// TIA Portal project "fill_level_inspector_1st_stage" (V17)

(* hardware
DEVICE "S7-1200 station_1"  S7-1200 Station
   slot 0: "Rack_0"  S7-1200 Rack  Rack  V1.0
   slot 1: "PLC_1"  CPU 1212C AC/DC/Rly  6ES7 212-1BE31-0XB0  V3.0
   slot 2: "DI 16x24VDC/DQ 16xRelay_1"  SM 1223 DI16/DQ16 x relay  6ES7 223-1PL32-0XB0  V2.0
DEVICE "HMI_1"  KTP600 Basic color PN
   slot 0: "HMI_1"  KTP600 Basic color PN  6AV6 647-0AD11-3AX0  12.0.0.0
   slot 1: "HMI_RT_1"  KTP600 Basic color PN  6AV6 647-0AD11-3AX0  12.0.0.0
   slot 5: "HMI_1.IE_CP_1"  PROFINET Interface  12.0.0.0
      slot 1: "PROFINET Interface_1"  PROFINET Interface
         slot 1: "Port_1"  Port
*)

// ===== PLC "PLC_1"  CPU 1212C AC/DC/Rly =====

VAR_GLOBAL   // PLC tag table "Default tag table"
   "START" AT %M0.0 : Bool;
   "STOP" AT %M0.1 : Bool;
   "SYSTEM_RUN" AT %M0.2 : Bool;
   "Bottle_Animation" AT %MW20 : Int;
   "Bottle_Output" AT %M50.0 : Bool;
   "Filling_Animation" AT %MW22 : Int;
   "Filling_Output" AT %M50.1 : Bool;
   "BottleFull_Animation" AT %MW24 : Int;
   "BottleFull_Output" AT %M50.2 : Bool;
   "Clock_Byte" AT %MB100 : Byte;
   "Clock_10Hz" AT %M100.0 : Bool;
   "Clock_5Hz" AT %M100.1 : Bool;
   "Clock_2.5Hz" AT %M100.2 : Bool;
   "Clock_2Hz" AT %M100.3 : Bool;
   "Clock_1.25Hz" AT %M100.4 : Bool;
   "Clock_1Hz" AT %M100.5 : Bool;
   "Clock_0.625Hz" AT %M100.6 : Bool;
   "Clock_0.5Hz" AT %M100.7 : Bool;
END_VAR

// folder: System blocks/Program resources

DATA_BLOCK "Counter_Bottle_Animation"   // DB1
{ S7_Optimized_Access := 'TRUE' }
AUTHOR : Simatic
FAMILY : IEC
NAME : CNTR
VERSION : 1.0
// stored: InstanceOfName IEC_COUNTER
"IEC_COUNTER"
BEGIN
END_DATA_BLOCK

DATA_BLOCK "Counter_Filling_Animation"   // DB4
{ S7_Optimized_Access := 'TRUE' }
AUTHOR : Simatic
FAMILY : IEC
NAME : CNTR
VERSION : 1.0
// stored: InstanceOfName IEC_COUNTER
"IEC_COUNTER"
BEGIN
END_DATA_BLOCK

DATA_BLOCK "Counter_BottleFull_Animation"   // DB5
{ S7_Optimized_Access := 'TRUE' }
AUTHOR : Simatic
FAMILY : IEC
NAME : CNTR
VERSION : 1.0
// stored: InstanceOfName IEC_COUNTER
"IEC_COUNTER"
BEGIN
END_DATA_BLOCK

// folder: (top level)

ORGANIZATION_BLOCK "Main"   // OB1, LAD, ProgramCycle
TITLE = "Main Program Sweep (Cycle)"
{ S7_Optimized_Access := 'TRUE' }
VERSION : 0.1
BEGIN

REGION Network 1: OPEN/CLOSE VALVE
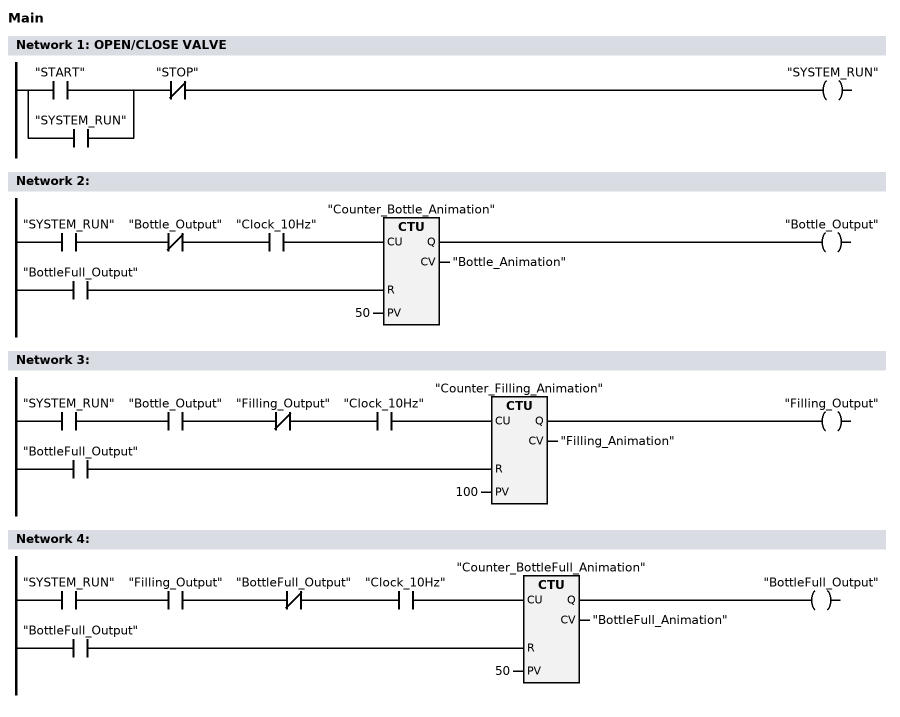
   RUNG wire#powerrail
      Contact( "START" )
      wire#w1
      I_Contact( "STOP" )
      Coil( "SYSTEM_RUN" )
   END_RUNG
   RUNG wire#powerrail
      Contact( "SYSTEM_RUN" )
   END_RUNG wire#w1
   // the same network as SCL:
   "SYSTEM_RUN" := ("START" OR "SYSTEM_RUN") AND NOT "STOP";
END_REGION

REGION Network 2
   "Counter_Bottle_Animation".CTU(CU := "SYSTEM_RUN" AND NOT "Bottle_Output" AND "Clock_10Hz",
                           R := "BottleFull_Output",
                           PV := 50,
                           CV => "Bottle_Animation");
   "Bottle_Output" := "Counter_Bottle_Animation".Q;
END_REGION

REGION Network 3
   "Counter_Filling_Animation".CTU(CU := "SYSTEM_RUN" AND "Bottle_Output" AND NOT "Filling_Output" AND "Clock_10Hz",
                           R := "BottleFull_Output",
                           PV := 100,
                           CV => "Filling_Animation");
   "Filling_Output" := "Counter_Filling_Animation".Q;
END_REGION

REGION Network 4
   "Counter_BottleFull_Animation".CTU(CU := "SYSTEM_RUN" AND "Filling_Output" AND NOT "BottleFull_Output" AND "Clock_10Hz",
                           R := "BottleFull_Output",
                           PV := 50,
                           CV => "BottleFull_Animation");
   "BottleFull_Output" := "Counter_BottleFull_Animation".Q;
END_REGION
END_ORGANIZATION_BLOCK

(* ===== HMI "HMI_RT_1" =====
system functions are stored by id; their names below are inferred from use
connection "HMI_Connection_1": ETHERNET, SMART_S7_1200_OMS

HMI tags "Default tag table"
   "START" : Bool = PLC START AT %M0.0, 1 s
   "STOP" : Bool = PLC STOP AT %M0.1, 1 s
   "SYSTEM_RUN" : Bool = PLC SYSTEM_RUN AT %M0.2, 1 s
   "Filling_Animation" : Int = PLC Filling_Animation AT %MW22, 1 s
   "BottleFull_Animation" : Int = PLC BottleFull_Animation AT %MW24, 1 s
   "Bottle_Animation" : Int = PLC Bottle_Animation AT %MW20, 1 s

screen "Screen_1" 320x240
   Button "Button_1" at 200,4 size 50x31; TextOff 'START'
      on Press: function_b14e0dd5("START", 0)
   Button "Button_2" at 258,3 size 50x31; TextOff 'STOP'
      on Press: function_b14e0dd5("STOP", 0)
   Circle "Circle_1" at 143,3 size 34x34
      Appearance <- "SYSTEM_RUN"
   GraphicView "Graphic view_1" at 3,176 size 314x40; Picture "probny_conveyer"
   GraphicView "Graphic view_3" at 34,111 size 26x82; Picture "glass_bottle_but_better"
      Visibility <- "Filling_Animation"
      HorizontalMovement <- "Bottle_Animation"
   GraphicView "Graphic view_2" at 86,111 size 26x82; Picture "glass_bottle_but_better"
      Visibility <- "Filling_Animation"
      HorizontalMovement <- "BottleFull_Animation"
   Rectangle "Rectangle_4" at 87,177 size 24x13
      Visibility <- "Filling_Animation"
      HorizontalMovement <- "BottleFull_Animation"
   Rectangle "Rectangle_5" at 87,164 size 24x13
      Visibility <- "Filling_Animation"
      HorizontalMovement <- "BottleFull_Animation"
   Rectangle "Rectangle_6" at 87,151 size 24x13
      Visibility <- "Filling_Animation"
      HorizontalMovement <- "BottleFull_Animation"
   Rectangle "Rectangle_7" at 87,138 size 24x13
      Visibility <- "Filling_Animation"
      HorizontalMovement <- "BottleFull_Animation"
   Ellipse "Ellipse_1" at 95,97 size 7x9
      Visibility <- "Filling_Animation"
*)